(* PLC project Unnamed, Unknown Unnamed 1 *)
(* stored: creationDateTime 2026-07-13T23:48:31, modificationDateTime 2026-07-13T23:48:31 *)

PROGRAM main

            for i := 0 to 10 do
    
end_for;
          
END_PROGRAM

CONFIGURATION Config0
  RESOURCE Res0 ON PLC
    TASK task0(INTERVAL := T#20ms, PRIORITY := 1);
    PROGRAM instance0 WITH task0 : main;
  END_RESOURCE
END_CONFIGURATION
